// LS Electric XG5000 project: Conveyer Controll with Button
// PLC LSPLC

PROGRAM NewProgram (task: 스캔 프로그램)

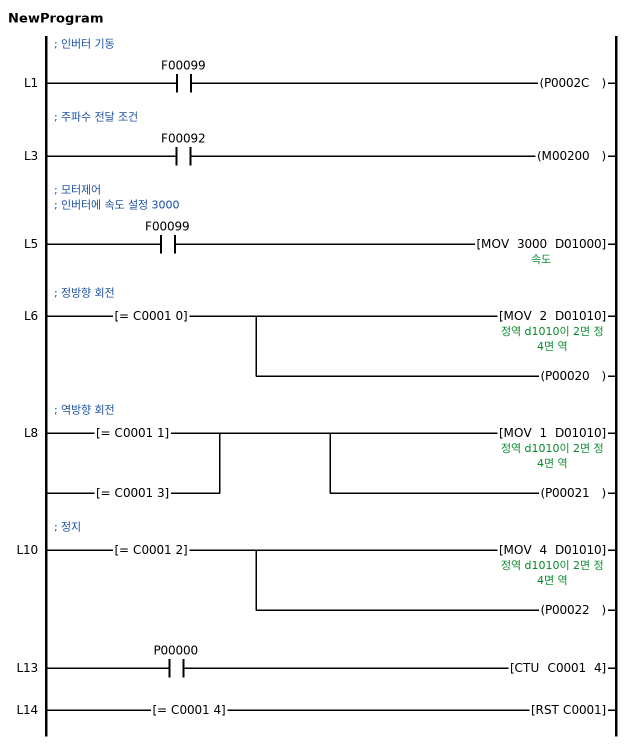
// 인버터 기동
; L1
LOAD      F00099
OUT       P0002C
// 주파수 전달 조건
; L3
LOAD      F00092
OUT       M00200
// 모터제어
; L5
LOAD      F00099
MOV       3000 D01000	// 속도
// output comment: 인버터에 속도 설정 3000
; L6
LOAD=     C0001 0
MOV       2 D01010	// 정역 d1010이 2면 정 4면 역
OUT       P00020
// output comment: 정방향 회전
; L8
LOAD=     C0001 1
OR=       C0001 3
MOV       1 D01010	// 정역 d1010이 2면 정 4면 역
OUT       P00021
// output comment: 역방향 회전
; L10
LOAD=     C0001 2
MOV       4 D01010	// 정역 d1010이 2면 정 4면 역
OUT       P00022
// output comment: 정지
; L13
LOAD      P00000
CTU       C0001 4
; L14
LOAD=     C0001 4
RST       C0001

VARIABLES AND COMMENTS (devices not used above)
D01020	WORD	가속
D01030	WORD	감속